//Enumeration for User Modes
TYPE E_PMLUserUnitMode : (
	ePMLUnitMode_Service		:=  4,
	ePMLUnitMode_Usermode2		:=  5,
	ePMLUnitMode_Usermode3		:=  6,
	ePMLUnitMode_Usermode4		:=  7,
	ePMLUnitMode_Usermode5 		:=  8,
	ePMLUnitMode_Usermode6 		:=  9,
	ePMLUnitMode_Usermode7 		:=  10
) DINT;
END_TYPE

(* stored: Version 1.1.0.1, ProductVersion 3.1.4024.12
   DUT E_PMLUserUnitMode: Id {d8b54365-f4c6-4f15-a178-811ad5541f6a} *)
